# EPICS StreamDevice protocol: rotating_sample_changerSup/rot_sample_changer.proto
Terminator = '\r';
ReplyTimeout = 2000;

getID {
    out "id";
    in "%/(.{0,39})/";
	ExtraInput = Ignore;
}

cmd {
    out "\$1";
}

setD {
    out "\$1 %d";
}
getD {
    out "\$1?";
    in "%d";
    ExtraInput = Ignore;
}
